FUNCTION_BLOCK FB_Totband
VAR_INPUT
	rTotband : REAL := 2;
	rPos : REAL;
END_VAR
VAR_OUTPUT
	rPosFilt : REAL := 0;
END_VAR
VAR
END_VAR

IF rPos > rTotband OR rPos < -rTotband THEN
	rPosFilt := rPos;
ELSE
	rPosFilt := 0;
END_IF

END_FUNCTION_BLOCK

(* stored: Version 1.1.0.1, ProductVersion 3.1.4024.12
   POU FB_Totband: Id {d9f76d3a-a277-4758-908c-b76ba2d94149}, SpecialFunc None *)
